TYPE ST_EcSlaveState :
STRUCT
	Device	: ST_EcDeviceState;	// Device state
	Link	: E_EcLinkState;	// Link state
END_STRUCT
END_TYPE

(* stored: Version 1.1.0.1, ProductVersion 3.1.4024.14
   DUT ST_EcSlaveState: Id {f60e2a48-970c-00ed-3e1d-7e3f68fd61d3} *)
